FUNCTION_BLOCK GrundstrukturObjekt IMPLEMENTS I_State
VAR_INPUT
	iMode				:INT;				// Information über aktuellen Betriebsmodi 
	iSkillCommand 		:INT;				// Steuerungsvariabel von Skill
	iSysCommand			:INT;				// Steuerungsvariabel von System
	iSysState			:INT;				// Information über Stand von System
	bReset				:BOOL;				// Trigger für Resett von Objekt
END_VAR
VAR_OUTPUT
	bDone				:BOOL;				// Information ob Skill ausgfeührt wurde
	bBusy				:BOOL;				// Information ob Skill im Moment ausgeführt wird
	bError				:BOOL;				// Information ob sich Skill in Fehlerzustand befindet
	iErrorID			:INT;				// Information um welchen Fehler es sich handelt	
END_VAR
VAR
	iState				:SkillState;		// Information über Zustand von Skill
END_VAR

PROPERTY P_State : INT
GET
P_State := iState;
END_GET
END_PROPERTY

END_FUNCTION_BLOCK

(* stored: Version 1.1.0.1
   POU GrundstrukturObjekt: Id {9e0cb548-32a9-47c1-a7f8-3617636e4541}, SpecialFunc None
   Property P_State: Id {052ef2e5-d2c5-42a0-9b3c-d98a0aaf411a}
   Get Get: Id {20cfde82-d3ed-4a74-ac63-78a27fed707b} *)
